FUNCTION_BLOCK ValveControlledCylinder
VAR_INPUT
	uDcvEnable : BOOL; 
	uDcv : LREAL;
	ReturnPressure : LREAL;
	SupplyPressure : LREAL;
	par : ST_pValveControlledCylinder;
	xPiston : LREAL;
	vPiston : LREAL;
END_VAR
VAR_OUTPUT
	F_Hydraulic : LREAL;
END_VAR
VAR
	PressurepA : LREAL;
	PressurepB : LREAL;
	
	y_tmp1 : LREAL;
	y_tmp2 : LREAL;
	F_Stribeck_Friction : LREAL;

//Pressure pA
fbPressureGradient_pA : PressureGradient;
//PressurepA : LREAL;

//Pressure pB
fbPressureGradient_pB : PressureGradient;
//PressurepB : LREAL;

//OrificeEquation QA and QB
fbOrificeEquationQ_P_A : OrificeEquation;
fbOrificeEquationQ_B_R : OrificeEquation;
fbOrificeEquationQ_P_B : OrificeEquation;
fbOrificeEquationQ_A_R : OrificeEquation;	
FlowQ_P_A : LREAL;
FlowQ_B_R : LREAL;	
FlowQ_P_B : LREAL;
FlowQ_A_R : LREAL;
FlowQA : LREAL;
FlowQB : LREAL;
FlowQL : LREAL := 0.00001;

//Control
ValveOpeningControl : LREAL := 0.0;
pVelocity : LREAL;

//BulkModulus
fbBulkModulus : BulkModulus;
fbVariableBulkModulus : VariableBulkModulus;

PistonArea : LREAL;
AnnulusArea : LREAL;

//ValveDynamics
fbValveDynamics : ValveDynamics;
uDcvDynamic : LREAL;


END_VAR


//IF uDcvEnable THEN
//	ValveOpeningControl := uDcv;
//ELSE 
//	ValveOpeningControl := 0;
//END_IF

	
PistonArea := EXPT(par.DBore,2) * (par.pi/4.0);
AnnulusArea := (EXPT(par.DBore,2) - EXPT(par.DRod,2)) * (par.pi/4.0);

//ValveOpeningControl := XboxControl.joyLeft;      Commented out xbox control as for now

//ValveDynamics
IF uDcvEnable THEN
	fbValveDynamics(
		udcv_IN := uDcv,
		DynamicValve => ValveOpeningControl
		);
ELSE
	fbValveDynamics(
		udcv_IN := 0,
		DynamicValve => ValveOpeningControl
		);	
END_IF

//VariableBulkModulus
fbVariableBulkModulus(
	OilBulkModulus := par.OilBulkModulus,
	AdiatricAirConstant := par.AdiatricAirConstant,
	AtmosphericPressure := par.AtmosphericPressure,
	VolumetricAirContentOfOil := par.VolumetricAirConstant
	);

//Pressure Gradient pA and Pressure pA
fbPressureGradient_pA(
	TotalVolume := par.VA0 + (xPiston * PistonArea),
	BulkModulus := fbBulkModulus.BulkModulus,
	FlowrateIn := FlowQA,
	FlowrateOut := (vPiston * PistonArea),
	p0 := par.pA0,
	param := par,
	Pressure => PressurepA		
	);

//Pressure Gradient pB and Pressure pB
fbPressureGradient_pB(
	TotalVolume := par.VB0 + ((par.xMax - xPiston) * AnnulusArea),
	BulkModulus := fbBulkModulus.BulkModulus,
	FlowrateIn := (vPiston * AnnulusArea),
	FlowrateOut := FlowQB + FlowQL,
	p0 := par.pB0,
	param := par,
	Pressure => PressurepB		
	);

//Flow through orifices Q_P_A, Q_A_R, Q_B_R, Q_P_B
fbOrificeEquationQ_P_A(
	PressureOut := PressurepA, 			
	PressureIn := SupplyPressure,	
	ValveOpening := ValveOpeningControl,	
	param := par,
	OrificeFlow => FlowQ_P_A
	);
	
fbOrificeEquationQ_A_R(
	PressureOut := ReturnPressure, 			
	PressureIn :=  PressurepA,	
	ValveOpening := ValveOpeningControl,	
	param := par,
	OrificeFlow => FlowQ_A_R
	);

fbOrificeEquationQ_B_R(
	PressureOut := ReturnPressure, 			
	PressureIn := PressurepB,			
	ValveOpening := ValveOpeningControl,
	param := par,
	OrificeFlow => FlowQ_B_R
	);
	
fbOrificeEquationQ_P_B(
	PressureOut := PressurepB, 			
	PressureIn := SupplyPressure,			
	ValveOpening := ValveOpeningControl,
	param := par,
	OrificeFlow => FlowQ_P_B
	);	

IF ValveOpeningControl > 0 THEN
	FlowQA := FlowQ_P_A;		
	FlowQB := FlowQ_B_R;
ELSIF ValveOpeningControl < 0 THEN
	FlowQA := FlowQ_A_R;		
	FlowQB := FlowQ_P_B;
ELSE
	FlowQA := 0.0;		
	FlowQB := 0.0;	
END_IF

// Hydraulic Force [N] //
//// Stribeck Friction Force [N] // Dette går til Urealistisk visualisator
//y_tmp1 := EXP((ABS(vPiston) * par.FrictionForceApproximationConstant) * 2.0);
//y_tmp2 := (y_tmp1 - 1.0) / (y_tmp1 + 1.0);
//F_Stribeck_Friction := (((EXP(( -(vPiston * y_tmp2)) / par.StaticFrictionTimeConstant) * ABS(par.StaticFrictionForce)) + par.ColoumbFriction) * y_tmp2) + (vPiston * par.ViscousFrictionCoefficient);
F_Hydraulic := PressurepA * PistonArea - PressurepB * AnnulusArea;  //F_Stribeck_Friction;
	
//PistonForce Cylinder
//fbPistonForce(
//	PressureBoreSide := PressurepA,
//	PressureRodSide := PressurepB,
//	Aa := PistonArea,
//	Ab := AnnulusArea,
//	PistonPosition := xPiston,
//	PistonVelocity := vPiston,
//	F_Piston => PistonForce
//	);

END_FUNCTION_BLOCK

(* stored: Version 1.1.0.1, ProductVersion 3.1.4024.9
   POU ValveControlledCylinder: Id {c1915dd1-7c80-44ad-a4db-c25faf141489}, SpecialFunc None *)
